(* IEC 61131-3 sources: Universal/UNIVERSAL/Interfaces/UNIVERSAL/Device1/Terminal1 (part 2) *)

FUNCTION Upgrade_1_ENTER
	// Upgrade.En_Read:= TRUE;
    Upgrade.Check_Upgrade:= TRUE;
END_FUNCTION

FUNCTION Upgrade_1_PRG
    IF (Upgrade.En_FirmWare) THEN
        Upgrade.En_Upgrade:= TRUE;
        GotoMask(Upgrade_Progress);
    ELSE
        Upgrade_1_ENTER();
    END_IF;
END_FUNCTION

(*				BEGIN IMPORT CODE				*)

FUNCTION NetMap_ENTER

    CurSlave:=      CurPosition;
    CurSlaveShow:=  TRUE;   // сообщаем стратегии что сейчас будем показывать текущего ведомого

	GotoMaskID(32); //SlaveState

END_FUNCTION

FUNCTION SlaveState_ESC
    CurSlaveShow:=  FALSE;// сообщаем стратегии что прекращаем показывать текущего ведомого
    IF (GetAlarmsCount() > 0) THEN
        SetLedStatus(12,1);// возвращаем управление колокольчиком основной программе
    ELSE
        SetLedStatus(12,0);
    END_IF;
    GotoMask(NetMap);
END_FUNCTION

FUNCTION Incr_REAL_x1000
    __TMP_REAL := __TMP_REAL + TO_REAL(__SYSVA_KEY_COUNTER)*1000.0;
    CheckLimitsDecr();
END_FUNCTION

FUNCTION Decr_REAL_x1000
    __TMP_REAL := __TMP_REAL - TO_REAL(__SYSVA_KEY_COUNTER)*1000.0;
    CheckLimitsDecr();
END_FUNCTION

(*				END IMPORT CODE					*)

FUNCTION DeviceRole_Class_PRG
    IF (StatePRG = STATE_PRG_READY) THEN
        StoreMask();
        StatePRG:= STATE_PRG_ON;
        NextCycleAction:= 2;
    ELSIF (StatePRG = STATE_PRG_ON) THEN
        Compare();
        IF (temp_Role <> Role) THEN
            IF (temp_Role = 0)OR(Role_Master) THEN
                (*Reboot_Reason:= 3;// изменение роли устройства
                StoreMask();
                GotoMask(NeedReboot);*)
                ShowPopUpQuestion(4); // изменение роли устройства
            ELSE
                Role:=      temp_Role;
                StoreMask();
                StatePRG:= STATE_PRG_READY;
                NextCycleAction:=   1;
            END_IF;
        ELSE
            StoreMask();
            StatePRG:= STATE_PRG_READY;
            NextCycleAction:=   1;
        END_IF;
    END_IF;
END_FUNCTION

FUNCTION DeviceRole_Class_ENTER
    IF (StatePRG <> STATE_PRG_READY) THEN
	    Compare();
        IF (temp_Role <> Role) THEN
            IF (temp_Role = 0)OR(Role_Master) THEN
                ShowPopUpQuestion(4);// изменение роли устройства
            ELSE
                Role:=  temp_Role;
            END_IF;
        END_IF;
    END_IF;
END_FUNCTION

FUNCTION HeatType_ENTER
	Compare ();
    IF (temp_HeatType <> HeatType) THEN
        IF (temp_HeatType = 1) OR (HeatType = 1)  THEN
            ShowPopUpQuestion(3);// изменение типа нагрева
        ELSE
            HeatType:= temp_HeatType;
        END_IF;
    END_IF;
END_FUNCTION

// Тест. Управление частотником
FUNCTION Main_Testing_ESC
    IF (EnPwdChgM) THEN
	    En_Testing:= TRUE;
        GotoLoop(TESTING);
        StatePRG:= STATE_PRG_READY;
    END_IF;
END_FUNCTION

FUNCTION Testing_ESC
    En_Testing:= FALSE;
	GotoMain();
    StatePRG:= STATE_PRG_OFF;
END_FUNCTION

// ModBus
FUNCTION Show_ports
    IF (Temp_MB_port = 0) THEN
        En_MB_Ethernet:= FALSE;
        En_MB_BMS_Card:= FALSE;
        En_MB_BMS2:= FALSE;
        En_MB_BMS:= FALSE;
    ELSIF (Temp_MB_port = 1) THEN
        En_MB_Ethernet:= TRUE;
        En_MB_BMS_Card:= FALSE;
        En_MB_BMS2:= FALSE;
        En_MB_BMS:= FALSE;
    ELSIF (Temp_MB_port = 2) THEN
        En_MB_Ethernet:= FALSE;
        En_MB_BMS_Card:= TRUE;
        En_MB_BMS2:= FALSE;
        En_MB_BMS:= TRUE;
        Temp_MB_Baudrate:= BMS_Card.Baudrate;
        Temp_MB_StopBits:= BMS_Card.StopBits;
        Temp_MB_Parity:= BMS_Card.Parity;
    ELSIF (Temp_MB_port = 3) THEN
        En_MB_Ethernet:= FALSE;
        En_MB_BMS_Card:= FALSE;
        En_MB_BMS2:= TRUE;
        En_MB_BMS:= TRUE;
        Temp_MB_Baudrate:= BMS2.Baudrate;
        Temp_MB_StopBits:= BMS2.StopBits;
        Temp_MB_Parity:= BMS2.Parity;
    END_IF;
END_FUNCTION

FUNCTION Port_Sel_ENTER
    IF (Temp_MB_port <> TO_USINT(__TMP_BYTE)) THEN
        Compare();
	    Show_ports();
    ELSE
        GotoNextField();
    END_IF;
END_FUNCTION

FUNCTION MB_Settings_1_PRG
    IF (StatePRG = STATE_PRG_READY) THEN
        StoreMask();
        StatePRG:= STATE_PRG_ON;
        NextCycleAction:=   1;
    ELSIF (StatePRG = STATE_PRG_ON) THEN
        Compare();
        IF (Temp_MB_port <> MB_port)
            OR (Temp_MB_Address <> MB_Address)
            OR ((Temp_MB_port = 2)AND (Temp_MB_Baudrate <> BMS_Card.Baudrate))
            OR ((Temp_MB_port = 2)AND (Temp_MB_StopBits <> BMS_Card.StopBits))
            OR ((Temp_MB_port = 2)AND (Temp_MB_Parity <> BMS_Card.Parity))
            OR ((Temp_MB_port = 3)AND (Temp_MB_Baudrate <> BMS2.Baudrate))
            OR ((Temp_MB_port = 3)AND (Temp_MB_StopBits <> BMS2.StopBits))
            OR ((Temp_MB_port = 3)AND (Temp_MB_Parity <> BMS2.Parity))
            THEN
            (*Reboot_Reason:= 4;// изменение настроек ModBus
            StoreMask();
            GotoMask(NeedReboot);*)
            ShowPopUpQuestion(5);// изменение настроек ModBus
        ELSE
            Show_ports();
            StatePRG:= STATE_PRG_READY;
            NextCycleAction:=   1;
        END_IF;
    END_IF;
END_FUNCTION

FUNCTION MB_Settings_1_ESC
    IF (StatePRG = STATE_PRG_READY) THEN
        GlobalEsc();
    ELSIF (StatePRG = STATE_PRG_ON) THEN
        Compare();
        IF (Temp_MB_port <> MB_port)
            OR (Temp_MB_Address <> MB_Address)
            OR ((Temp_MB_port = 2)AND (Temp_MB_Baudrate <> BMS_Card.Baudrate))
            OR ((Temp_MB_port = 2)AND (Temp_MB_StopBits <> BMS_Card.StopBits))
            OR ((Temp_MB_port = 2)AND (Temp_MB_Parity <> BMS_Card.Parity))
            OR ((Temp_MB_port = 3)AND (Temp_MB_Baudrate <> BMS2.Baudrate))
            OR ((Temp_MB_port = 3)AND (Temp_MB_StopBits <> BMS2.StopBits))
            OR ((Temp_MB_port = 3)AND (Temp_MB_Parity <> BMS2.Parity))
            THEN
            (*Reboot_Reason:= 4;// изменение настроек ModBus
            StoreMask();
            GotoMask(NeedReboot);*)
            ShowPopUpQuestion(5);// изменение настроек ModBus
        ELSE
            GlobalEsc();
        END_IF;
    END_IF;
END_FUNCTION

FUNCTION Mul_DWORD_x2
    __TMP_DWORD := __TMP_DWORD * 2;
    CheckLimitsIncr();
END_FUNCTION

FUNCTION Div_DWORD_x2
    __TMP_DWORD := __TMP_DWORD / 2;
    CheckLimitsDecr();
END_FUNCTION
FUNCTION Upgrade_OS_ESC
	Upgrade.REQ_OS_upgrade:= FALSE;
    GotoLoop(UPGRADE);
END_FUNCTION

FUNCTION Upgrade_OS_PRG
	Upgrade.ANSW_OS_upgrade:= TRUE;
    GotoMask(Upgrade_Progress);
END_FUNCTION

FUNCTION PRG_button_goto10
	 IF (StatePRG = STATE_PRG_READY) THEN
        StoreMask();
        StatePRG:= STATE_PRG_ON;
        NextCycleAction:=   2;
    ELSIF (StatePRG = STATE_PRG_ON) THEN
        Compare();
        StatePRG:= STATE_PRG_READY;
        NextCycleAction:=   1;
    END_IF;
END_FUNCTION

// Переход на следующую маску в режиме программирования
FUNCTION DOWN_ENTER_Move
    IF (StatePRG = STATE_PRG_ON) THEN
        GotoNextMask();
        checkZeroColumn:= TRUE;
    END_IF;
END_FUNCTION

// Переход на предыдущую маску в режиме программирования
FUNCTION UP_ENTER_Move
    IF (StatePRG = STATE_PRG_ON) THEN
        GotoPreviousMask();
        checkZeroColumn:= TRUE;
    END_IF;
END_FUNCTION

FUNCTION Decrement // уменьшение байтовой переменной с индикацией стрелки
    Decrement_BYTE();
    downArrow:= TRUE;
END_FUNCTION

FUNCTION Increment  // увеличение байтовой переменной с индикацией стрелки
    Increment_BYTE();
    upArrow:=   TRUE;
END_FUNCTION

FUNCTION BoolDown   // уменьшение булевой переменной с индикацией стрелки
	BoolSwap();
    downArrow:= TRUE;
END_FUNCTION

FUNCTION BoolUp     // увеличение булевой переменной с индикацией стрелки
	BoolSwap();
    upArrow:=   TRUE;
END_FUNCTION

//FUNCTION FConfigSetBool  // принятие булевой переменной с индикацией выбора
    //MakeChoice:=        TRUE;
    //NextCycleAction:=   3;
//END_FUNCTION
//
//FUNCTION FConfigSetByte  // принятие байтовой переменной с индикацией выбора
    //Compare();
    //MakeChoice:=        TRUE;
    //NextCycleAction:=   3;
//END_FUNCTION
//
//FUNCTION FConfigSetPriority  // принятие  переменной ModeSEQ c переходом к петле CONFIRM_CONFIG
    //Compare();
    //NextCycleAction:=   6;
//END_FUNCTION
//
//
//FUNCTION FConfig_LastMask    // принятие последней в петле байтовой переменной с индикацией выбора
	//Compare();
    //MakeChoice:=        TRUE;
    //IF (IsPOOL) THEN
        //NextCycleAction:=   6;
    //ELSE
        //NextCycleAction:=   5;
    //END_IF;
//END_FUNCTION
//
//FUNCTION FConfig_ESC  // запрос на возврат к началу первой конфигурации
    //IF (CompletePreConfig) THEN
        //ShowPopUpQuestion(12);  // Выйти из мастера конфигураций
    //ELSE
        //StatePRG:= STATE_PRG_ALWAYS_ON;
        //MakeChoice:=    FALSE;
        //ShowPopUpQuestion(7);   // Вернуться к началу конфигурации?
    //END_IF;
//END_FUNCTION

FUNCTION SWAP_Sp100
    BoolSwap();
    IF (wCoil_Mode_A_B)AND(Par_Sp100) THEN
        ShowPopUpMessage(12, SHORT_POPUP_TIME);
        //Par_Sp100:=   FALSE;
    END_IF;
END_FUNCTION

FUNCTION SWAP_Tp10 // Проверка при переключении параметра Tp10 в меню
    BoolSwap();
    IF NOT(SNSR_Thru.Use)OR(SNSR_Thru.Error <> 10) THEN
		IF NOT(Par_Tp10)THEN
            ShowPopUpMessage(11, SHORT_POPUP_TIME);
            Par_Tp10:=   TRUE;
        END_IF;
    END_IF;
END_FUNCTION

FUNCTION ManualManager // Вход и выход из ручного режима
    VAR_INPUT
        in : BOOL;
    END_VAR

    IF (in)AND NOT(ManualManage)THEN
        ManualManage:=  TRUE;
        ShowPopUpMessage(15, SHORT_POPUP_TIME); //  Ручной режим включен
    ELSIF NOT(in)AND (ManualManage)THEN
        ManualManage:=  FALSE;
        CurRow:= 0;
        ShowPopUpMessage(16, SHORT_POPUP_TIME); // Ручной режим выключен
    END_IF;

END_FUNCTION

FUNCTION Param_UP   // Переход вверх

    IF (StatePRG = STATE_PRG_READY) THEN
        IF (CurRow > 1) THEN
            CurRow:= CurRow - 1;
        ELSE

            //MaskMng.shift_position:= -(TO_DINT(__SYSVA_KEY_COUNTER)/20) - 1;
            Position:= Position - TO_DINT(__SYSVA_KEY_COUNTER)/20 - 1;

            //IF (Position + MaskMng.shift_position < 1) THEN
                //__SYSVA_KEY_COUNTER:= 0;
                //CurRow:= num_Rows;
                //Beep();
            //END_IF;
            IF (Position < 1) THEN
                __SYSVA_KEY_COUNTER:= 0;
                Position:= cnt_Items - num_Rows + 1;
                CurRow:= num_Rows;
                //Beep();
            END_IF;
        END_IF;
        CurList_Position:= Position + CurRow - 1;
        Display.Hint:= Display.Descr[CurRow];
        update_ParamMenu_List:=      TRUE;
    ELSIF (StatePRG = STATE_PRG_ON) THEN

        CASE (Display.value_Storage[CurRow_modePRG]) OF
            0: // BOOL
                IF (Display.value_BOOL[CurRow_modePRG] = 2) THEN
                    Display.value_BOOL[CurRow_modePRG]:= 1;
                END_IF;
            1: // UINT
                Display.value_INT[CurRow_modePRG]:=  Display.value_INT[CurRow_modePRG] + TO_INT(__SYSVA_KEY_COUNTER);
            2: // REAL
                Display.value_REAL[CurRow_modePRG]:=  Display.value_REAL[CurRow_modePRG] + TO_REAL(__SYSVA_KEY_COUNTER)/10.0;
        END_CASE;
        CheckValueBorders ();
    END_IF;
    NextCycleAction:= 12; //Обновление подсказки и позиции
END_FUNCTION

FUNCTION Param_DOWN   // Переход вверх

    IF (StatePRG = STATE_PRG_READY) THEN
        IF (CurRow < num_Rows) THEN
            CurRow:= CurRow + 1;
        ELSE
            Position:= Position + TO_DINT(__SYSVA_KEY_COUNTER)/20 + 1;

            IF (Position > cnt_Items - num_Rows + 1) THEN
                __SYSVA_KEY_COUNTER:= 0;
                Position:= 1;
                CurRow:= 1;
                //Beep();
            END_IF;
           //MaskMng.shift_position:= TO_DINT(__SYSVA_KEY_COUNTER)/20 + 1;
            //
            //IF (Position + MaskMng.shift_position > cnt_Items - num_Rows + 1) THEN
                //__SYSVA_KEY_COUNTER:= 0;
                //CurRow:= 1;
                //Beep();
            //END_IF;
        END_IF;
        CurList_Position:= Position + CurRow - 1;
        Display.Hint:= Display.Descr[CurRow];
        update_ParamMenu_List:=      TRUE;
    ELSIF (StatePRG = STATE_PRG_ON) THEN

        CASE (Display.value_Storage[CurRow_modePRG]) OF
            0: // BOOL
                IF (Display.value_BOOL[CurRow_modePRG] = 1) THEN
                    Display.value_BOOL[CurRow_modePRG]:= 2;
                END_IF;
            1: // UINT
                Display.value_INT[CurRow_modePRG]:=  Display.value_INT[CurRow_modePRG] - TO_INT(__SYSVA_KEY_COUNTER);
            2: // REAL
                Display.value_REAL[CurRow_modePRG]:=  Display.value_REAL[CurRow_modePRG] - TO_REAL(__SYSVA_KEY_COUNTER)/10.0;
        END_CASE;
        CheckValueBorders ();
    END_IF;
    NextCycleAction:= 12; //Обновление подсказки и позиции
END_FUNCTION

FUNCTION Param_ENTER   // Подтверждение
    IF (StatePRG = STATE_PRG_ON) THEN

        Write_Parameter();

        IF (CurRow_modePRG < num_Rows) THEN
            CurRow_modePRG:= CurRow_modePRG + 1;
        ELSE
            Position:= Position + TO_DINT(__SYSVA_KEY_COUNTER)/20 + 1;

            IF (Position > cnt_Items - num_Rows + 1) THEN
                __SYSVA_KEY_COUNTER:= 0;
                Position:= 1;
                CurRow_modePRG:= 1;
                //Beep();
            END_IF;
        END_IF;
        //getParamMenu:=      TRUE;
        CurList_Position:= Position + CurRow_modePRG - 1;
        Display.Hint:= Display.Descr[CurRow_modePRG];
        update_ParamMenu_List:=      TRUE;
    END_IF;

    NextCycleAction:= 12; //Обновление подсказки и позиции
END_FUNCTION

FUNCTION Write_Parameter // Запись параметра

    CheckValueBorders ();
    CASE (Display.value_Storage[CurRow_modePRG]) OF
        0: // BOOL
            IF (Display.value_BOOL[CurRow_modePRG] = 1) THEN ;
                param.BOOL[Display.value_Address[CurRow_modePRG]]:= TRUE;
            ELSIF (Display.value_BOOL[CurRow_modePRG] = 2) THEN ;
                param.BOOL[Display.value_Address[CurRow_modePRG]]:= FALSE;
            END_IF;
        1: // INT
            IF (param.INT[Display.value_Address[CurRow_modePRG]] <>
                Display.value_INT[CurRow_modePRG])
            THEN
                //MaskMng.param_ChangeNotify:= Display.Descr[CurRow_modePRG];
                param.INT[Display.value_Address[CurRow_modePRG]]:= Display.value_INT[CurRow_modePRG];
            END_IF;
        2: // REAL
            IF (param.REAL[Display.value_Address[CurRow_modePRG]] <>
                Display.value_REAL[CurRow_modePRG])
            THEN
                //MaskMng.param_ChangeNotify:= Display.Descr[CurRow_modePRG];
                param.REAL[Display.value_Address[CurRow_modePRG]]:= Display.value_REAL[CurRow_modePRG];
            END_IF;
    END_CASE;

    MaskMng.param_ChangeNotify:= TO_USINT(Display.Descr[CurRow_modePRG]);
END_FUNCTION

FUNCTION Param_ESC   // Переход вверх

    IF (StatePRG = STATE_PRG_READY) THEN
        //cnt_Items:=  0;
        Position:=      1;
        autoHideArrowsOff:=     FALSE;
        GlobalEsc();
    ELSIF (StatePRG = STATE_PRG_ON) THEN
        StatePRG:=  STATE_PRG_READY;
        CurRow:= CurRow_modePRG;
        CurRow_modePRG:=    0;
        //getParamMenu:=      TRUE;
        update_ParamMenu_List:= TRUE;
    END_IF;

END_FUNCTION

FUNCTION CheckValueBorders   // Проверка границ значений

    CASE (Display.value_Storage[CurRow_modePRG]) OF
            0: // BOOL
               ;
            1: // UINT
                IF (Display.value_INT[CurRow_modePRG] < Display.value_MinINT[CurRow_modePRG]) THEN
                    Display.value_INT[CurRow_modePRG]:= Display.value_MaxINT[CurRow_modePRG];
                    Beep();
                ELSIF (Display.value_INT[CurRow_modePRG] > Display.value_MaxINT[CurRow_modePRG]) THEN
                    Display.value_INT[CurRow_modePRG]:= Display.value_MinINT[CurRow_modePRG];
                    Beep();
                END_IF;
            2: // REAL
                IF (Display.value_REAL[CurRow_modePRG] < Display.value_MinREAL[CurRow_modePRG]) THEN
                    Display.value_REAL[CurRow_modePRG]:= Display.value_MaxREAL[CurRow_modePRG];
                    Beep();
                ELSIF (Display.value_REAL[CurRow_modePRG] > Display.value_MaxREAL[CurRow_modePRG]) THEN
                    Display.value_REAL[CurRow_modePRG]:= Display.value_MinREAL[CurRow_modePRG];
                    Beep();
                END_IF;
        END_CASE;
END_FUNCTION

FUNCTION UpdateCurPos
// Отображение расширенного описания текущей позиции
    IF (ModePRG) THEN
        Display.Hint:= Display.Descr[CurRow_modePRG];
        CurList_Position:= Position + CurRow_modePRG - 1;
    ELSE
        Display.Hint:= Display.Descr[CurRow];
        CurList_Position:= Position + CurRow - 1;
    END_IF;
END_FUNCTION

FUNCTION CheckListBorders   // Проверка границ списка
    //VAR
        //lastPixelPosition : USINT; // позиция последнего пикселя
    //END_VAR;
//
    //IF (Position <= 1) THEN
        //upArrow:= FALSE;
    //ELSE
        //upArrow:= TRUE;
    //END_IF;
//
    //IF (Position >= cnt_Items - num_Rows + 1) OR
       //(cnt_Items < num_Rows)
    //THEN
        //downArrow:= FALSE;
    //ELSE
        //downArrow:= TRUE;
    //END_IF;

(*
    IF (Slider_Height = 0) THEN
        Slider_Height:= TO_USINT(48 / cnt_Items);
    END_IF;

    lastPixelPosition:= Slider_Height * TO_USINT(Position);

    IF (lastPixelPosition <= 8) THEN
        Slider_1:= lastPixelPosition;
    ELSIF (lastPixelPosition <= 16) THEN
        Slider_2:= lastPixelPosition - 8;
        IF (Slider_Height > 8) THEN
             Slider_1:= 16 - (Slider_Height - (16 - lastPixelPosition)) ;
        END_IF;
    END_IF;
*)
END_FUNCTION

FUNCTION Param_PRG   //

    //StoreMask();

    IF (StatePRG = STATE_PRG_READY) THEN        // вход в режим редактирования
            //150121 2.7.6.0 Запрет для пользователя упразднен, т.к. скрываются все ненужные пункты меню.
            //IF (UnitOn)AND(PwdTyp < 2) THEN         //  Для пользователя изменения во время работы запрещены
            //    ShowPopUpMessage(1, POPUP_TIME);    //  Выключите установку для изменения настроек!
            //ELSE
                StatePRG:=  STATE_PRG_ON;
                CurRow_modePRG:= CurRow;
                CurRow:=    0;
                // getParamMenu:=      TRUE;
                update_ParamMenu_List:= TRUE;
                NextCycleAction:= 12; //Обновление подсказки и позиции
            //END_IF;

    ELSIF (StatePRG = STATE_PRG_ON) THEN        // выход из режима редактирования

        Write_Parameter();

        StatePRG:=  STATE_PRG_READY;
        CurRow:= CurRow_modePRG;
        CurRow_modePRG:=    0;
        //getParamMenu:=      TRUE;
        update_ParamMenu_List:= TRUE;
        NextCycleAction:= 12; //Обновление подсказки и позиции
    END_IF;
END_FUNCTION

//FUNCTION GoToConfiguration
	////load_Config:= TRUE;
    ////isConfigMenu:= TRUE;
    ////getConfigMenu:= TRUE;
    ////CurRow:=            1;
    ////CurRow_modePRG:=    0;
    ////cnt_Items:= 0;
    ////GotoMask(LoadConfig_Mask);
    //ConfigMng.checkConfigFile:= TRUE;
//END_FUNCTION

FUNCTION ConfigMenu_UP   // Переход вверх
    IF (CurRow > 1) THEN
        CurRow:= CurRow - 1;
    ELSE
        Position:= Position - TO_DINT(__SYSVA_KEY_COUNTER)/20 - 1;

        IF (Position < 1) THEN
            __SYSVA_KEY_COUNTER:= 0;
            Position:= cnt_Items - num_Rows + 1;
            CurRow:= num_Rows;
            //Beep();
        END_IF;

        IF (isConfigMenu) THEN
            getConfigMenu:= TRUE;
        ELSE
            getParamMenu:= TRUE;
        END_IF;
    END_IF;

    CurList_Position:= Position + CurRow - 1;
    Display.Hint:= Display.Descr[CurRow];
END_FUNCTION

FUNCTION ConfigMenu_DOWN   // Переход вниз
    IF (CurRow < num_Rows) THEN
        CurRow:= CurRow + 1;
    ELSE
        Position:= Position + TO_DINT(__SYSVA_KEY_COUNTER)/20 + 1;

        IF (Position > cnt_Items - num_Rows + 1) THEN
            __SYSVA_KEY_COUNTER:= 0;
            Position:= 1;
            CurRow:= 1;
            //Beep();
        END_IF;

        IF (isConfigMenu) THEN
            getConfigMenu:= TRUE;
        ELSE
            getParamMenu:= TRUE;
        END_IF;
    END_IF;

    CurList_Position:= Position + CurRow - 1;
    Display.Hint:= Display.Descr[CurRow];
END_FUNCTION

FUNCTION ConfigMenu_ENTER   //
    IF (Display.value_BOOL[CurRow] = 4) // каталог
    THEN
        //IF (CurLevel < 10) THEN
            //Display.Path.MenuPoint[CurLevel]:= CurMenuPoint;
            //Display.Path.Position[CurLevel]:= Position;
            //Display.Path.Row[CurLevel]:= CurRow;
            //CurLevel:= CurLevel + 1;
            SaveMenuPos();
            CurMenuPoint:= TO_DINT(Display.Descr[CurRow]);
            getConfigMenu:= TRUE;
        //END_IF;
        IF (CurLevel < 10) THEN
            CurRow:=            1;
            Position:=          1;
            CurList_Position:=  1;
        END_IF;
    ELSIF (Display.value_BOOL[CurRow] = 7) // действие?
    THEN
        //Display.Path.MenuPoint[CurLevel]:= CurMenuPoint;
        //Display.Path.Position[CurLevel]:= Position;
        //Display.Path.Row[CurLevel]:= CurRow;
        SaveMenuPos();
        CurMenuPoint:= TO_DINT(Display.Descr[CurRow]);
        getConfigMenu:= TRUE;
    ELSE
        Display.Path.MenuPoint[CurLevel]:= CurMenuPoint;
        Display.Path.Position[CurLevel]:= Position;
        Display.Path.Row[CurLevel]:= CurRow;
        CurMenuPoint:= TO_DINT(Display.Descr[CurRow]);
        setConfigItem:= TRUE;
    END_IF;
    //NextCycleAction:= 12;
    Display.Hint:= Display.Descr[CurRow];
END_FUNCTION

FUNCTION ConfigMenu_ESC   //
    IF (CurLevel > ConfigStartLevel) THEN
        LoadMenuPos();
    ELSE
        //Перебрасываем в начало конфигуратора
        Position:=          1;
        CurMenuPoint:=      0;
        CurList_Position:=  1;
        CurRow:=            1;

        //IF (CurMenuPoint <> 0) THEN
            //Position:= 1;
            //CurMenuPoint:= 0;
            //CurList_Position:= 1;
            //CurRow:= 1;
        //ELSE
            //IF (ConfigStartLevel <> 0) THEN
                //IF (IsConfigChanged) THEN
                    ////Сохранить конфигурацию?
                    //ShowPopUpQuestion(21); //InstantAction:=  255; //DF_CFG_END
                //ELSE
                    //GlobalEsc();
                //END_IF;
            //END_IF;
        //END_IF;
    END_IF;

    getConfigMenu:= TRUE;
    //cnt_Items:=  0;

    //NextCycleAction:= 12;
END_FUNCTION

FUNCTION Signal_DOWN

    CASE CurRow OF
        1:
            mask_List_pos:=  mask_List_pos + TO_DINT(__SYSVA_KEY_COUNTER)/20 + 1;

            IF (mask_List_pos > cnt_Items) THEN
                __SYSVA_KEY_COUNTER:= 0;
                mask_List_pos:= 1;
                Beep();
            END_IF;

            Display.Descr[1]:= mask_List[mask_List_pos];
            Display.Hint:= mask_List_Sec[mask_List_pos];
            //Display.Hint:= Display.Descr[1];
            ConfigMng.recount_Types:= TRUE;
            recount_IO:= TRUE;
            getMinMax:= TRUE;

        2:
           (*Сдвиг окна позиции*)
			ConfigMng.mask_IO_List_pos:= ConfigMng.mask_IO_List_pos + TO_DINT(__SYSVA_KEY_COUNTER)/20 + 1;
			(*Проверка выхода за границы*)
			IF (ConfigMng.mask_IO_List_pos > ConfigMng.cnt_IO_Items) THEN
                __SYSVA_KEY_COUNTER:= 0;
                ConfigMng.mask_IO_List_pos:= 0;
                Beep();
            END_IF;

			Display.Descr[2]:= TO_UINT(ConfigMng.mask_IO_List[ConfigMng.mask_IO_List_pos]);
            //Display.Descr[3]:= TO_USINT(ConfigMng.mask_IO_List_pos);
            //IF (ConfigMng.mask_IO_List_pos = 0) THEN
                //Display.Hint:= 0;
            //ELSE
                //Display.Hint:= ConfigMng.mask_IO_List[0] + 1;
            //END_IF;

        3:
            (*Сдвиг окна позиции*)
			ConfigMng.mask_TypeList_pos:= ConfigMng.mask_TypeList_pos - TO_DINT(__SYSVA_KEY_COUNTER)/20 - 1;
			(*Проверка выхода за границы*)
			IF (ConfigMng.mask_TypeList_pos < 0) THEN
                __SYSVA_KEY_COUNTER:= 0;
                ConfigMng.mask_TypeList_pos:= ConfigMng.cnt_TypeItems - 1;
                Beep();
            END_IF;

			Display.Descr[3]:= TO_UINT(ConfigMng.mask_TypeList[ConfigMng.mask_TypeList_pos]);

        4:
            Display.value_REAL[4]:= Display.value_REAL[4] - TO_REAL(__SYSVA_KEY_COUNTER/20) - 1.0;
            IF (Display.value_REAL[4] < Display.value_MinREAL[4]) THEN
                Display.value_REAL[4]:= Display.value_MaxREAL[4];
                Beep();
            END_IF;

        5:
            Display.value_REAL[5]:= Display.value_REAL[5] - TO_REAL(__SYSVA_KEY_COUNTER/20) - 1.0;
            IF (Display.value_REAL[5] < Display.value_MinREAL[5]) THEN
                Display.value_REAL[5]:= Display.value_MaxREAL[5];
                Beep();
            END_IF;
    END_CASE;
END_FUNCTION

FUNCTION Signal_UP

    CASE CurRow OF
        1:
            mask_List_pos:=  mask_List_pos - TO_DINT(__SYSVA_KEY_COUNTER)/20 - 1;

            IF (mask_List_pos < 1) THEN
                __SYSVA_KEY_COUNTER:= 0;
                mask_List_pos:= cnt_Items;
                Beep();
            END_IF;
            //getIOConfig:= TRUE;

            Display.Descr[1]:= mask_List[mask_List_pos];
            Display.Hint:= mask_List_Sec[mask_List_pos];
            //Display.Descr[2]:= ConfigMng.mask_IO_List[0];
            //Display.Hint:= Display.Descr[1];
            ConfigMng.recount_Types:= TRUE;
            recount_IO:= TRUE;
            getMinMax:= TRUE;

        2:
           (*Сдвиг окна позиции*)
			ConfigMng.mask_IO_List_pos:= ConfigMng.mask_IO_List_pos - TO_DINT(__SYSVA_KEY_COUNTER)/20 - 1;
			(*Проверка выхода за границы*)
			IF (ConfigMng.mask_IO_List_pos < 0) THEN
                __SYSVA_KEY_COUNTER:= 0;
                ConfigMng.mask_IO_List_pos:= ConfigMng.cnt_IO_Items;
                Beep();
            END_IF;

			Display.Descr[2]:= TO_UINT(ConfigMng.mask_IO_List[ConfigMng.mask_IO_List_pos]);
            //Display.Descr[3]:= TO_USINT(ConfigMng.mask_IO_List_pos);
            //IF (ConfigMng.mask_IO_List_pos = 0) THEN
                //Display.Hint:= 0;
            //ELSE
                //Display.Hint:= ConfigMng.mask_IO_List[0] + 1;
            //END_IF;

        3:
            (*Сдвиг окна позиции*)
			ConfigMng.mask_TypeList_pos:= ConfigMng.mask_TypeList_pos + TO_DINT(__SYSVA_KEY_COUNTER)/20 + 1;
			(*Проверка выхода за границы*)
			IF (ConfigMng.mask_TypeList_pos > ConfigMng.cnt_TypeItems - 1) THEN
                __SYSVA_KEY_COUNTER:= 0;
                ConfigMng.mask_TypeList_pos:= 0;
                Beep();
            END_IF;

			Display.Descr[3]:= TO_UINT(ConfigMng.mask_TypeList[ConfigMng.mask_TypeList_pos]);

        4:
            Display.value_REAL[4]:= Display.value_REAL[4] + TO_REAL(__SYSVA_KEY_COUNTER/20) + 1.0;
            IF (Display.value_REAL[4] > Display.value_MaxREAL[4]) THEN
                Display.value_REAL[4]:= Display.value_MinREAL[4];
                Beep();
            END_IF;

        5:
            Display.value_REAL[5]:= Display.value_REAL[5] + TO_REAL(__SYSVA_KEY_COUNTER/20) + 1.0;
            IF (Display.value_REAL[5] > Display.value_MaxREAL[5]) THEN
                Display.value_REAL[5]:= Display.value_MinREAL[5];
                Beep();
            END_IF;

    END_CASE;
END_FUNCTION

FUNCTION Signal_ESC

    //RestoreMask();
    GlobalEsc();

    //CurLevel:= CurLevel - 1;
    //CurMenuPoint:=  Display.Path.MenuPoint[CurLevel];
    //Position:= Display.Path.Position[CurLevel];
    //CurRow:= Display.Path.Row[CurLevel];
    //Display.Path.MenuPoint[CurLevel]:= 0;
    //CurList_Position:= Position + CurRow - 1;

    //getConfigMenu:= TRUE;

END_FUNCTION

FUNCTION Signal_ENTER

    CASE CurRow OF
        1:
            recount_IO:= TRUE;
            //IF (ConfigMng.mask_IO_List_pos = 0) THEN
                //Display.Hint:= 0;
            //ELSE
                //Display.Hint:= ConfigMng.mask_IO_List[0] + 1;
            //END_IF;

            IF (num_Rows = 2) THEN
                CurRow:= 2;
            ELSE
                CurRow:= 3;
                Display.Descr[3]:= TO_UINT(ConfigMng.mask_TypeList[ConfigMng.mask_TypeList_pos]);
            END_IF;
        2:
            ConfigMng.setIoItem:= TRUE;
            //Display.Hint:= 0;
            CurRow:= 1;
        3:
            recount_IO:= TRUE;
            CASE Display.Descr[3] OF
                5,6,7,8,9: //AI с min/max
                    CurRow:= 4;
            ELSE
                CurRow:= 2;
            END_CASE;
            getMinMax:= TRUE;
        4:
            //сделать запись в переменную Min для сигнала
            ConfigMng.setMinMax:= TRUE;
            CurRow:= 5;
        5:
            //сделать запись в переменную Max для сигнала
            ConfigMng.setMinMax:= TRUE;
            CurRow:= 2;
    END_CASE;

END_FUNCTION

// Управление маской Control_Mode------------
FUNCTION Control_Mode_UP
	upArrow:= TRUE;
    IF (temp_Mode_Control > 1) THEN
        temp_Mode_Control:= temp_Mode_Control - 1;
    ELSE
        temp_Mode_Control:= 10;
    END_IF;

    IF (IsPOOL)(*OR(IsICE)*) THEN
        IF (temp_Mode_Control = 10) THEN
            temp_Mode_Control:= 8;
        ELSIF (temp_Mode_Control = 6) OR (temp_Mode_Control = 5) THEN
            temp_Mode_Control:= 4;
        ELSIF (temp_Mode_Control = 3) THEN
            temp_Mode_Control:= 2;
        END_IF;
    END_IF;
END_FUNCTION

FUNCTION Control_Mode_DOWN
	downArrow:= TRUE;
    IF (temp_Mode_Control < 10) THEN
        temp_Mode_Control:= temp_Mode_Control + 1;
    ELSE
        temp_Mode_Control:= 1;
    END_IF;

    IF (IsPOOL)(*OR(IsICE)*) THEN
        IF (temp_Mode_Control = 3) THEN
            temp_Mode_Control:= 4;
        ELSIF (temp_Mode_Control = 5) OR (temp_Mode_Control = 6) THEN
            temp_Mode_Control:= 7;
        ELSIF (temp_Mode_Control = 9) OR (temp_Mode_Control = 10) THEN
            temp_Mode_Control:= 1;
        END_IF;
    END_IF;
END_FUNCTION

FUNCTION Control_Mode_ENTER
	Mode_Control:= temp_Mode_Control;
END_FUNCTION
//-------------------------------------------

// Управление маской Schedule_Manage------------
FUNCTION Schedule_Manage_UP
	upArrow:= TRUE;
    temp_En_Schedule:= NOT(temp_En_Schedule);
END_FUNCTION

FUNCTION Schedule_Manage_DOWN
	downArrow:= TRUE;
    temp_En_Schedule:= NOT(temp_En_Schedule);
END_FUNCTION

FUNCTION Schedule_Manage_ENTER
	En_Schedule:= temp_En_Schedule;
END_FUNCTION

//-------------------------------------------

//FUNCTION Load_Config
    //load_Config:= TRUE;
    //GotoMask(LoadConfig_Mask);
//END_FUNCTION

// Управление масками вх/вых -------------------------------------
FUNCTION IO_DOWN
    IF (StatePRG = STATE_PRG_ON) THEN
        IF (CurRow = 3) THEN // Надпись Режим
            IF (Display.value_BOOL[1] = 1) THEN //руч.
                CurRow:= 4;
            ELSE
                IF  (Display.MaskID = 11) OR // Дискретные входы
                    (Display.MaskID = 14)    // Аналоговые выходы
                THEN
                    CurRow:= 5;
                ELSE
                    Beep();
                END_IF;
            END_IF;
        ELSIF (CurRow = 4) THEN // Надпись Статус
            CurRow:= 3;
        ELSIF (CurRow = 5) THEN // Надпись инверсия
            CurRow:= 3;
        ELSIF (CurRow_modePRG = 3) THEN // Изменение режима
            IF (Display.value_BOOL[1] = 0) THEN
                 Display.value_BOOL[1]:= 1;
            ELSIF( Display.value_BOOL[1] = 1) THEN
                Display.value_BOOL[1]:= 0;
            END_IF;
            //MaskMng.ValueWasChanged:= TRUE;
        ELSIF (CurRow_modePRG = 4) THEN // Изменение значения
            CASE Display.MaskID OF
                11, 13:(*Digital*)
                    Display.value_BOOL[2]:= 2; //OFF
                    MaskMng.ValueWasChanged:= TRUE;
                12:(*Analog inputs*)
                    IF (Display.En_RealValue[1]) THEN
                        Display.value_REAL[1]:= Display.value_REAL[1] - TO_REAL(__SYSVA_KEY_COUNTER)/10.0;
                        IF (Display.value_REAL[1] < Display.value_MinREAL[1]) THEN
                            Display.value_REAL[1]:= Display.value_MaxREAL[1];
                            __SYSVA_KEY_COUNTER:= 0;
                            Beep();
                        END_IF;
                    ELSIF (Display.En_IntValue[1]) THEN
                        Display.value_INT[1]:= Display.value_INT[1] - TO_INT(__SYSVA_KEY_COUNTER)/10 - 1;
                        IF (Display.value_INT[1] < Display.value_MinINT[1]) THEN
                            Display.value_INT[1]:= Display.value_MaxINT[1];
                            __SYSVA_KEY_COUNTER:= 0;
                            Beep();
                        END_IF;
                    END_IF;
                    //MaskMng.ValueWasChanged:= TRUE;

                14:
                    Display.value_REAL[1]:= Display.value_REAL[1] - TO_REAL(__SYSVA_KEY_COUNTER)/10.0;
                    IF (Display.value_REAL[1] < 0.0) THEN
                        Display.value_REAL[1]:= 0.0;
                        Beep();
                    END_IF;
            END_CASE;
        ELSIF (CurRow_modePRG = 5) THEN // Изменение инверсии
            IF (Display.value_BOOL[3] = 0) THEN
                Display.value_BOOL[3]:= 1;
            ELSE
                Display.value_BOOL[3]:= 0;
            END_IF;
        END_IF;
    ELSE
        mask_List_pos:=  mask_List_pos + TO_DINT(__SYSVA_KEY_COUNTER)/20 + 1;
        IF (mask_List_pos > cnt_Items) THEN
            __SYSVA_KEY_COUNTER:= 0;
            mask_List_pos:= 1;
            Beep();
        END_IF;
        Display.Descr[1]:= TO_UINT(cfgIO.Link_toCodes[TO_DINT(mask_List[mask_List_pos])]) - TO_UINT(MaskMng.sig_start) + 1;
        Display.Descr[2]:= mask_List[mask_List_pos];
    END_IF;
END_FUNCTION

FUNCTION IO_UP
    IF (StatePRG = STATE_PRG_ON) THEN
        IF (CurRow = 3) THEN // Надпись Режим
            IF (Display.value_BOOL[1] = 1) THEN //руч.
                CurRow:= 4;
            ELSE
                IF  (Display.MaskID = 11) OR // Дискретные входы
                    (Display.MaskID = 14)    // Аналоговые выходы
                THEN
                    CurRow:= 5;
                ELSE
                    Beep();
                END_IF;
            END_IF;
        ELSIF (CurRow = 4) THEN // Надпись Статус
            CurRow:= 3;
        ELSIF (CurRow = 5) THEN // Надпись инверсия
            CurRow:= 3;
        ELSIF (CurRow_modePRG = 3) THEN // Изменение режима
            IF (Display.value_BOOL[1] = 0) THEN
                 Display.value_BOOL[1]:= 1;
            ELSIF( Display.value_BOOL[1] = 1) THEN
                Display.value_BOOL[1]:= 0;
            END_IF;
            //MaskMng.ValueWasChanged:= TRUE;
        ELSIF (CurRow_modePRG = 4) THEN // Изменение значения
            CASE Display.MaskID OF
                11, 13:(*Digital*)
                    Display.value_BOOL[2]:= 1; //ON
                    MaskMng.ValueWasChanged:= TRUE;
                12:(*Analog inputs*)
                    IF (Display.En_RealValue[1]) THEN
                        Display.value_REAL[1]:= Display.value_REAL[1] + TO_REAL(__SYSVA_KEY_COUNTER)/10.0;
                        IF (Display.value_REAL[1] > Display.value_MaxREAL[1]) THEN
                            Display.value_REAL[1]:= Display.value_MinREAL[1];
                            __SYSVA_KEY_COUNTER:= 0;
                            Beep();
                        END_IF;
                    ELSIF (Display.En_IntValue[1]) THEN
                        Display.value_INT[1]:= Display.value_INT[1] + TO_INT(__SYSVA_KEY_COUNTER)/10 + 1;
                        IF (Display.value_INT[1] > Display.value_MaxINT[1]) THEN
                            Display.value_INT[1]:= Display.value_MinINT[1];
                            __SYSVA_KEY_COUNTER:= 0;
                            Beep();
                        END_IF;
                    END_IF;

                14: (*Analog outputs*)
                    Display.value_REAL[1]:= Display.value_REAL[1] + TO_REAL(__SYSVA_KEY_COUNTER)/10.0;
                    IF (Display.value_REAL[1] > 10.0) THEN
                        Display.value_REAL[1]:= 10.0;
                        Beep();
                    END_IF;
            END_CASE;
        ELSIF (CurRow_modePRG = 5) THEN // Изменение инверсии
            IF (Display.value_BOOL[3] = 1) THEN
                Display.value_BOOL[3]:= 0;
            ELSE
                Display.value_BOOL[3]:= 1;
            END_IF;
        END_IF;
    ELSE
        mask_List_pos:=  mask_List_pos - TO_DINT(__SYSVA_KEY_COUNTER)/20 - 1;
        IF (mask_List_pos < 1) THEN
            __SYSVA_KEY_COUNTER:= 0;
            mask_List_pos:= cnt_Items;
            Beep();
        END_IF;
        Display.Descr[1]:= TO_UINT(cfgIO.Link_toCodes[TO_DINT(mask_List[mask_List_pos])]) - TO_UINT(MaskMng.sig_start) + 1;
        Display.Descr[2]:= mask_List[mask_List_pos];
    END_IF;
END_FUNCTION

FUNCTION IO_PRG
    IF (StatePRG = STATE_PRG_READY) THEN        // вход в режим редактирования
        StatePRG:=  STATE_PRG_ON;
        CurRow:= 3;
        CurRow_modePRG:= 0;
    ELSIF (StatePRG = STATE_PRG_ON) THEN        // выход из режима редактирования
        StatePRG:=  STATE_PRG_READY;
        CurRow:= 0;
        CurRow_modePRG:= 0;
        MaskMng.ValueWasChanged:= TRUE;
    ELSIF (StatePRG = STATE_PRG_OFF) THEN        //ручной режим недоступен
        ShowPopUpMessage(17, SHORT_POPUP_TIME);
    END_IF;
END_FUNCTION

FUNCTION IO_ENTER
     IF (StatePRG = STATE_PRG_ON) THEN  // ручное управление
        IF (CurRow <> 0) THEN           // Пункты
           // IF (mask_List[mask_List_pos] >= 64) AND (mask_List[mask_List_pos] <= 83) THEN
            //    Beep();
            //ELSE          // НЕ DP-TOP
                CurRow_modePRG:= CurRow;
                CurRow:= 0;
           // END_IF;
        ELSIF (CurRow_modePRG = 3) THEN // Режим
            CurRow:= CurRow_modePRG;
            CurRow_modePRG:= 0;
            MaskMng.ValueWasChanged:= TRUE;
        ELSIF (CurRow_modePRG = 4) THEN // Статус
            CurRow:= CurRow_modePRG;
            CurRow_modePRG:= 0;
            MaskMng.ValueWasChanged:= TRUE;
        ELSIF (CurRow_modePRG = 5) THEN // Инверсия
            CurRow:= CurRow_modePRG;
            CurRow_modePRG:= 0;
            MaskMng.ValueWasChanged:= TRUE;
        END_IF;
    END_IF;
END_FUNCTION
//---------------------------------------------------------------

// Управление маской коррекции -------------------------------------
FUNCTION CORR_DOWN

    IF (StatePRG = STATE_PRG_ON) THEN
        (*Analog inputs correction*)
        IF (Display.En_RealValue[1]) THEN
            //Display.value_REAL[1]:= Display.value_REAL[1] - TO_REAL(__SYSVA_KEY_COUNTER)/10.0;
            Display.value_REAL[1]:= Display.value_REAL[1] - Display.value_REAL[8];
            IF (Display.value_REAL[1] < Display.value_MinREAL[1]) THEN
                Display.value_REAL[1]:= Display.value_MaxREAL[1];
                __SYSVA_KEY_COUNTER:= 0;
                Beep();
            END_IF;
        ELSIF (Display.En_IntValue[1]) THEN
            //Display.value_INT[1]:= Display.value_INT[1] - TO_INT(__SYSVA_KEY_COUNTER)/10 - 1;
            Display.value_INT[1]:= Display.value_INT[1] - Display.value_INT[8];
            IF (Display.value_INT[1] < Display.value_MinINT[1]) THEN
                Display.value_INT[1]:= Display.value_MaxINT[1];
                __SYSVA_KEY_COUNTER:= 0;
                Beep();
            END_IF;
        END_IF;
    ELSE
        mask_List_pos:=  mask_List_pos + TO_DINT(__SYSVA_KEY_COUNTER)/20 + 1;
        IF (mask_List_pos > cnt_Items) THEN
            __SYSVA_KEY_COUNTER:= 0;
            mask_List_pos:= 1;
            Beep();
        END_IF;
        Display.Descr[1]:= TO_UINT(cfgIO.Link_toCodes[TO_DINT(mask_List[mask_List_pos])]) - TO_UINT(MaskMng.sig_start) + 1;
        Display.Descr[2]:= mask_List[mask_List_pos];
    END_IF;

END_FUNCTION

FUNCTION CORR_UP

    IF (StatePRG = STATE_PRG_ON) THEN
        (*Analog inputs correction*)
        IF (Display.En_RealValue[1]) THEN
            //Display.value_REAL[1]:= Display.value_REAL[1] + TO_REAL(__SYSVA_KEY_COUNTER)/10.0;
            Display.value_REAL[1]:= Display.value_REAL[1] + Display.value_REAL[8];
            IF (Display.value_REAL[1] > Display.value_MaxREAL[1]) THEN
                Display.value_REAL[1]:= Display.value_MinREAL[1];
                __SYSVA_KEY_COUNTER:= 0;
                Beep();
            END_IF;
        ELSIF (Display.En_IntValue[1]) THEN
            //Display.value_INT[1]:= Display.value_INT[1] + TO_INT(__SYSVA_KEY_COUNTER)/10 + 1;
            Display.value_INT[1]:= Display.value_INT[1] + Display.value_INT[8];
            IF (Display.value_INT[1] > Display.value_MaxINT[1]) THEN
                Display.value_INT[1]:= Display.value_MinINT[1];
                __SYSVA_KEY_COUNTER:= 0;
                Beep();
            END_IF;
        END_IF;
    ELSE
        mask_List_pos:=  mask_List_pos - TO_DINT(__SYSVA_KEY_COUNTER)/20 - 1;
        IF (mask_List_pos < 1) THEN
            __SYSVA_KEY_COUNTER:= 0;
            mask_List_pos:= cnt_Items;
            Beep();
        END_IF;
        Display.Descr[1]:= TO_UINT(cfgIO.Link_toCodes[TO_DINT(mask_List[mask_List_pos])]) - TO_UINT(MaskMng.sig_start) + 1;
        Display.Descr[2]:= mask_List[mask_List_pos];
    END_IF;

END_FUNCTION

FUNCTION CORR_PRG
    IF (StatePRG = STATE_PRG_READY) THEN        // вход в режим редактирования
        StatePRG:=  STATE_PRG_ON;
        CurRow:= 0;
        CurRow_modePRG:= 3;
    ELSIF (StatePRG = STATE_PRG_ON) THEN        // выход из режима редактирования
        StatePRG:=  STATE_PRG_READY;
        CurRow:= 0;
        CurRow_modePRG:= 0;
        MaskMng.ValueWasChanged:= TRUE;
    ELSIF (StatePRG = STATE_PRG_OFF) THEN        //ручной режим недоступен
        ShowPopUpMessage(17, SHORT_POPUP_TIME);
    END_IF;
END_FUNCTION

FUNCTION CORR_ENTER
    IF (StatePRG = STATE_PRG_ON) THEN  // ручное управление
        MaskMng.ValueWasChanged:= TRUE;
    END_IF;
END_FUNCTION
//---------------------------------------------------------------
//----------------------- Main Menu -----------------------------
FUNCTION MainMenu_DOWN   // Переход вниз

    IF (CurRow < num_Rows) THEN
        Display.UoM[CurRow]:= Display.UoM[CurRow] - 1;
        CurRow:= CurRow + 1;
        Display.UoM[CurRow]:= Display.UoM[CurRow] + 1;
    ELSE
        Position:= Position + TO_DINT(__SYSVA_KEY_COUNTER)/20 + 1;

        IF (Position > cnt_Items - num_Rows + 1) THEN
            __SYSVA_KEY_COUNTER:= 0;
            Position:= 1;
            CurRow:= 1;
            //Beep();
        END_IF;
        update_MainMenu_List:= TRUE;
    END_IF;

    CurList_Position:= Position + CurRow - 1;
END_FUNCTION

FUNCTION MainMenu_UP   // Переход вверх

    IF (CurRow > 1) THEN
        Display.UoM[CurRow]:= Display.UoM[CurRow] - 1;
        CurRow:= CurRow - 1;
        Display.UoM[CurRow]:= Display.UoM[CurRow] + 1;
    ELSE
        Position:= Position - TO_DINT(__SYSVA_KEY_COUNTER)/20 - 1;

        IF (Position < 1) THEN
            __SYSVA_KEY_COUNTER:= 0;
            Position:= cnt_Items - num_Rows + 1;
            CurRow:= num_Rows;
            //Beep();
        END_IF;
        update_MainMenu_List:= TRUE;
    END_IF;

    CurList_Position:= Position + CurRow - 1;
END_FUNCTION

FUNCTION MainMenu_ENTER   //

    IF (Display.value_Type[CurRow] = 0) // каталог
    THEN
        IF (CurLevel < 10) THEN
            SaveMenuPos();
            //CurLevel:= CurLevel + 1;
            CurMenuPoint:= TO_DINT(Display.Descr[CurRow]);
            getMainMenu:= TRUE;
        END_IF;
        CurRow:= 1;
        Position:= 1;
    ELSIF (Display.value_Type[CurRow] = 1) // переход на  другую маску
    THEN
        //CurMenuPoint:= Display.Descr[CurRow];
        //getMainMenu:= TRUE;
        SaveMenuPos();
        //CurLevel:= CurLevel + 1;
        GotoMaskID(TO_USINT(Display.value_MinINT[CurRow]), TO_USINT(Display.value_MaxINT[CurRow]));
        Display.UoM[1]:= 0;
        Display.UoM[2]:= 0;
        Display.UoM[3]:= 0;
        Display.Descr[1]:= 0;
        Display.Descr[2]:= 0;
        Display.Descr[3]:= 0;
        CurRow:= 0;
    ELSIF (Display.value_Type[CurRow] = 2) // всплывающие окна
    THEN
        SaveMenuPos();
        GotoMaskID(TO_USINT(Display.value_MinINT[CurRow]), TO_USINT(Display.value_MaxINT[CurRow]));
    END_IF;
    CurList_Position:= 1;
END_FUNCTION

FUNCTION MainMenu_ESC   //
    IF (CurLevel > 1) THEN
        LoadMenuPos();
        getMainMenu:= TRUE;
    ELSE
        GlobalEsc();
    END_IF;
END_FUNCTION

//---------------------------------------------------------------
FUNCTION GotoMaskID
//Загрузка маски или петли по MaskID с сохранением пути
    VAR_INPUT
        iMaskID : USINT;
    END_VAR

    StoreMaskID();
    LoadMaskID(iMaskID, 0);
END_FUNCTION

FUNCTION GotoMaskID
//Загрузка маски или петли по MaskID с сохранением пути
    VAR_INPUT
        iMaskID : USINT;
        iParam : USINT; // передаваемый параметр
    END_VAR

    StoreMaskID();
    LoadMaskID(iMaskID, iParam);
END_FUNCTION

FUNCTION LoadMaskID
//Загрузка маски или петли по MaskID
    VAR_INPUT
        iMaskID : USINT;
        iParam : USINT; // передаваемый параметр
    END_VAR

    Display.MaskID:= TO_UINT(iMaskID);

    CASE iMaskID OF
        1: // Гл.экран	DF_MID_MAIN
            //GotoLoop(MAIN);
            GotoMask(Main_Mask);
            //При выходе в гл.меню или на гл.экран система возвращается в работу
            SystemPause:= FALSE;

        2: // Логин	DF_MID_LOGIN
            PwdIn := 0;                 // Reset password
            IncrTmp := 0;
            PwdRes := 0;
            CleanPwd();
            GotoMask(Pwd_LogIn);

        3: // Осн.меню	DF_MID_MMENU
            MainMenuVisibility_Is_Set:= FALSE;
	        ParamVisibility_Is_Set:= 	FALSE;

            getMainMenu:= TRUE;
            StatePRG:= STATE_PRG_OFF;
            GotoMask(Menu_Main);
            //При выходе в гл.меню или на гл.экран система вовзвращается в работу
            SystemPause:= FALSE;

        4: // Управление	DF_MID_ONOFF
            IF (LocalMode = 0)AND(Role_Slave) THEN
                StatePRG:= STATE_PRG_READY;// режим до редактирования
            ELSE
                StatePRG:= STATE_PRG_ALWAYS_ON;// режим редактирования
            END_IF;
            GotoLoop(ONOFF);

        5: // Маска загрузки	DF_MID_LOAD
            IF (UnitOff) THEN
                MaskMng.LoadMaskMode:= iParam;

                IF (iParam = 0) THEN //Загрузка при выходе из конфигуратора
                    ConfigMng.checkConfigFile:= TRUE;
                ELSIF (iParam = 1) THEN //Загрузка при входе в конфигуратор
                    ConfigMng.checkConfigFile:= TRUE;
                ELSIF (iParam = 2) THEN   //Загрузка конфигуратора из конфигуратора
                    //CurLevel:= ConfigStartLevel; возвращаемся к началу конфигуратора
                    //CurList_Position:= 1;
                   IsConfigChanged:= TRUE;
                    load_Config:= TRUE;
                ELSIF (iParam = 3) THEN   //Сохранение конфигуратора без выхода
                    save_Config:= TRUE;
                ELSIF (iParam = 4) THEN   //Сохранение конфигуратора с выходом
                    save_Config:= TRUE;
                END_IF;

                GotoMask(LoadConfig_Mask);
            ELSE
                ShowPopUpMessage(1, POPUP_TIME, TRUE);//  Выключите установку для изменения настроек!
            END_IF;
        6: //Настройки Ethernet DF_MID_ETH
            read_EthernetSettings:= TRUE;
            StatePRG:= STATE_PRG_READY;
            GotoMask(EthernetConfig_Mask);

        7: // Управление расписанием	DF_MID_SCH_MG
            temp_En_Schedule:= En_Schedule;
            StatePRG:= STATE_PRG_ON;
            GotoMask (Schedule_Manage);

        8: // Журнал аварий	DF_MID_ALOG
            gotoAlarmLog();

        9: // Последовательности	DF_MID_SEQ
            GotoLoop(SEQUENCES);

        10: // Мастер конфигурации	DF_MID_CFG_M
            IF (iParam = 1) THEN
                CurMenuPoint:=  0;
                Position:= 1;
                CurList_Position:= 1;
                CurRow:= 1;
                CurRow_modePRG:=    0;
                ConfigStartLevel:= CurLevel;
            END_IF;

            getConfigMenu:= TRUE;
            GotoMask(REF_CONFIGURATOR);

        11: //Дискретные входы	DF_MID_IO_DI
            CurRow:=            1;
            CurRow_modePRG:=    0;
            getIOList:=         TRUE;
            IF (UnitOn) THEN
                StatePRG:= STATE_PRG_OFF;
            ELSE
                StatePRG:= STATE_PRG_READY;
            END_IF;
            GotoMask(IO_DI);

        12: //Аналоговые входы	DF_MID_IO_AI
            CurRow:=            1;
            CurRow_modePRG:=    0;
            getIOList:=         TRUE;
            IF (UnitOn) THEN
                StatePRG:= STATE_PRG_OFF;
            ELSE
                StatePRG:= STATE_PRG_READY;
            END_IF;
            GotoMask(IO_AI);

        13: //Дискретные выходы	DF_MID_IO_DO
            CurRow:=            1;
            CurRow_modePRG:=    0;
            getIOList:=         TRUE;
            IF (UnitOn) THEN
                StatePRG:= STATE_PRG_OFF;
            ELSE
                StatePRG:= STATE_PRG_READY;
            END_IF;
            GotoMask(IO_DO);

        14: //Аналоговые выходы	DF_MID_IO_AO
            CurRow:=            1;
            CurRow_modePRG:=    0;
            getIOList:=         TRUE;
            IF (UnitOn) THEN
                StatePRG:= STATE_PRG_OFF;
            ELSE
                StatePRG:= STATE_PRG_READY;
            END_IF;
            GotoMask(IO_AO);

        15: //Уставка	DF_MID_SET
            getParam:= TRUE;
            IF (LocalMode = 0)AND(Role_Slave) THEN
                StatePRG:= STATE_PRG_READY;// режим до редактирования
            ELSE
                StatePRG:= STATE_PRG_ALWAYS_ON;// режим редактирования
            END_IF;
            GotoLoop(SET);

        16: //Выход	DF_MID_OUT
            GotoMask(Pwd_LogOut);

        17: //Роль устройства	DF_MID_GROLE
            temp_Role:= Role;
            StatePRG:= STATE_PRG_ALWAYS_ON;
            Gotomask(DeviceRole);
            GotoCursor (0,10);// кидаем за пределы экрана. ТОЛЬКО ДЛЯ 1 IO переменной на экране! Использовать Compare() без NextField!

        18: //Настройки группы	DF_MID_GSET
            IF (Role_Master) THEN
                IF (Num_Slaves > 0) THEN
                    CurSlave:=  1;
                    CurSlaveShow:=  TRUE;
                    StatePRG:= STATE_PRG_READY;// режим готовности к редактированию
                    GotoMask (SlaveSet);
                ELSE
                    ShowPopUpMessage(6, POPUP_TIME, TRUE);//  Состав группы не объявлен!
                END_IF;
            ELSE
                StatePRG:= STATE_PRG_ON;// режим готовности к редактированию
                Gotomask(LocalSet);// если ведомый - местные настройки (выбор режима)
                GotoCursor(0,10);
            END_IF;

        19: //Состав группы	DF_MID_GSTCT
            IF (Role_Master) THEN
                StatePRG:= STATE_PRG_ALWAYS_ON;// режим редактирования сразу
                Gotomask(GroupStructure);// если мастер-переходим к выбору состава группы
                GotoCursor (0,10);// кидаем за пределы экрана. ТОЛЬКО ДЛЯ 1 IO переменной на экране! Использовать Compare() без NextField!
           ELSE
                ShowPopUpMessage(2, POPUP_TIME, TRUE);//  Для доступа, выберите роль устройства: ВЕДУЩИЙ // если ведомый - заглушка
           END_IF;

        20: // Маска параметров	DF_MID_PAR
            //setParamMask(TO_USINT(Display.value_MaxINT[CurRow]));
            CurParam:=          iParam;
            getParamMenu:=      TRUE;
            cnt_Items:=         0;
            StatePRG:=          STATE_PRG_READY;
            GotoMask(REF_Parameters);

        21: //ХМ: Статистика	DF_MID_CM_STA
            //Show_CompStats:= TRUE;
            Display.Index:=     -1;
            StatePRG:=          STATE_PRG_READY;
            GotoLoop(FRIDGE_STATS);

        22: // Дата и время	DF_MID_DTIME
            StatePRG:=          STATE_PRG_READY;
            GotoLoop(DATETIME);

        23: //Язык	DF_MID_LANG
            StatePRG:=          STATE_PRG_ALWAYS_ON;
            Gotomask(Language);

        24: //Управление доступом	DF_MID_PASS
            IncrTmp :=          0;
            StatePRG:=          STATE_PRG_READY;
            GotoMask(PWDCHG);

        25: //Коррекция датчиков	DF_MID_SCORR
            MaskMng.getCorrList:= TRUE;
            StatePRG:= STATE_PRG_READY;
            GotoMask(CORR_AI);

        26: //Настройки ModBus	DF_MID_MODBUS
            IF (is_TOP) THEN
                ShowPopUpMessage(9, POPUP_TIME, TRUE);//  Доступно только со шкафа управления!
            // 20.07.20 v.2.6.0.0
            //ELSIF (IsDLE)AND(Role_Slave) THEN
            //    ShowPopUpMessage(10, POPUP_TIME, TRUE);//  Доступно только с ВЕДУЩЕГО!
            ELSE
                IF (Ethernet.Protocol[1] = 4) OR (Ethernet.Protocol[1] = 5) THEN
                    MB_port:= 1;
                ELSIF (BMS_card.Protocol = 4) OR (BMS_card.Protocol = 5) THEN
                    MB_port:= 2;
                ELSIF (BMS2.Protocol = 4) OR (BMS2.Protocol = 5) THEN
                    MB_port:= 3;
                ELSE
                    MB_port:= 0;
                END_IF;
                Temp_MB_port:= MB_port;
                Temp_MB_Address:= MB_Address;
                Show_ports();
                StatePRG:= STATE_PRG_READY;
                GotoLoop(MODBUS);
            END_IF;

        27: //Обновление	DF_MID_UPGR
            IF (UnitOff) THEN
                IF (iParam = 1) THEN //USB
                    IF (isUSB) THEN
                        Upgrade.UpgradeDrive:= 1; //SYS_DISK_USB
                        Upgrade.Check_Upgrade:= TRUE;
                        StatePRG:= STATE_PRG_ALWAYS_ON;
                        NextCycleAction:= 4; // GotoLoop (UPGRADE);
                    ELSE
                        //Вставьте USB-накопитель
                        ShowPopUpMessage(24, SHORT_POPUP_TIME, TRUE);
                    END_IF;
                ELSE
                    Upgrade.UpgradeDrive:= 0; //SYS_DISK_INTERNAL
                    Upgrade.Check_Upgrade:= TRUE;
                    StatePRG:= STATE_PRG_ALWAYS_ON;
                    NextCycleAction:= 4; // GotoLoop (UPGRADE);
                END_IF;
            ELSE
                ShowPopUpMessage(1, POPUP_TIME, TRUE);//  Выключите установку для изменения настроек!
            END_IF;

        28: //Расписание	DF_MID_SCH
            IF (is_TOP) THEN
                ShowPopUpMessage(9, POPUP_TIME, TRUE);//  Доступно только со шкафа управления!
            ELSIF (IsDLE)AND(Role_Slave) THEN
                ShowPopUpMessage(10, POPUP_TIME, TRUE);//  Доступно только с ВЕДУЩЕГО!
            ELSE
                StatePRG:= STATE_PRG_READY;
                GotoLoop (SCHEDULE);
            END_IF;

        29: //Режим управления	DF_MID_CMOD
            IF (is_TOP) THEN
                ShowPopUpMessage(9, POPUP_TIME, TRUE);//  Доступно только со шкафа управления!
            ELSIF (IsDLE)AND(Role_Slave)AND NOT(LocalMode) THEN
                ShowPopUpMessage(10, POPUP_TIME, TRUE);//  Доступно только с ВЕДУЩЕГО!
            ELSE
                temp_Mode_Control:= Mode_Control;
                StatePRG:= STATE_PRG_ON;
                GotoLoop (CONTROL_MODE);
            END_IF;

        30: //Маска сообщения	DF_MID_MSG
            ;

        31: //Маска вопроса	DF_MID_QSTN
            ReturnToPrevMask:= TRUE;
            StatePRG:= STATE_PRG_OFF;
            DTPopUp:= 0; //без таймера всплывающего окна
            PopUp_Question:= iParam;
            Gotomask(PopUp_Question_Mask);

        32: //Маска ведомых   DF_MID_SLST
            MaskMng.setStatePRG:= TRUE;
            GotoLoop(SLAVESTATES);

        33: //Роль устройства	DF_MID_ROLE
            temp_Role:= Role;
            StatePRG:= STATE_PRG_ALWAYS_ON;// режим редактирования сразу
            GotoLoop(UNITCONFIG);
            GotoCursor (0,10);// кидаем за пределы экрана. ТОЛЬКО ДЛЯ 1 IO переменной на экране! Использовать Compare() без NextField!

        34: //Настройки BMS   DF_MID_BMS
            IF (Role_Slave)OR(is_TOP) THEN
                Temp_MB_Baudrate:= BMS2.Baudrate;
                Temp_MB_Parity:= BMS2.Parity;
                Temp_MB_StopBits:= BMS2.StopBits;
            ELSE
                Temp_MB_Baudrate:= FBus2.Baudrate;
                Temp_MB_Parity:= FBus2.Parity;
                Temp_MB_StopBits:= FBus2.StopBits;
            END_IF;
            En_MB_BMS:= TRUE;
            StatePRG:= STATE_PRG_READY;//
            GotoLoop(BMS_SETTINGS);

         35: //Загрузка/Сохранение на USB DF_MID_PARMNG
            IF (isUSB) THEN
                Display.Hint:= TO_UINT(iParam);
                IF (iParam = 1) THEN
                    ShowPopUpQuestion(23, TRUE); //Сохранить параметры на USB?
                ELSE
                    ShowPopUpQuestion(22, TRUE); //Загрузить параметры с USB?
                END_IF;
            ELSE
                ShowPopUpMessage(24, SHORT_POPUP_TIME, TRUE); //Вставьте USB-накопитель
            END_IF;

         36: //Дискретные входы (конфиг) DF_MID_CFG_DI
            Position:= 1;
            CurRow:= 1;
            cnt_Items:= 0;
            getIOConfig:= TRUE;

            GotoMask(CFG_DI);

         37: //Аналоговые входы (конфиг) DF_MID_CFG_AI
            Position:= 1;
            CurRow:= 1;
            cnt_Items:= 0;
            getIOConfig:= TRUE;

            GotoMask(CFG_AI);

         38: //Дискретные выходы (конфиг) DF_MID_CFG_DO
            Position:= 1;
            CurRow:= 1;
            cnt_Items:= 0;
            getIOConfig:= TRUE;

            GotoMask(CFG_DO);

         39: //Аналоговые выходы (конфиг) DF_MID_CFG_AO
            Position:= 1;
            CurRow:= 1;
            cnt_Items:= 0;
            getIOConfig:= TRUE;

            GotoMask(CFG_AO);

         40: //Холодильная машина DF_MID_COLM
            StatePRG:= STATE_PRG_OFF;
            GotoLoop(FRIDGE);

         41: //Карта сети DF_MID_NETM
            StatePRG:= STATE_PRG_OFF;
            IF (Role_Master) THEN // для мастера
                IF (Num_Slaves > 0) THEN
                    Gotomask(NetMap);
                    IF (CurPosition = 0)OR(CurPosition > Num_Slaves) THEN
                        CurPosition:=   1;// в первую позицию, если впервые. Остальные запоминаем
                    END_IF;
                    CurShow[CurPosition]:=  TRUE;
                ELSE
                    ShowPopUpMessage(6, POPUP_TIME); //Состав группы не объявлен!
                END_IF;
            ELSE // для ведомых
                Gotomask(MasterState);
            END_IF;

        42: //Информация DF_MID_INFO
            GotoLoop(INFO);

        43: //Набор уставок	DF_MID_PSET
            getParam:= TRUE;
            StatePRG:= STATE_PRG_ALWAYS_ON;// режим редактирования
            GotoLoop(PRESETS);
            GotoCursor(0, 10);

        44: //Пароувлажнитель DF_MID_HUMID
            GotoLoop(HUMID);

        45: //Настройки соединения DF_MID_RESSET
            StatePRG:=              STATE_PRG_READY;
            MaskMng.get_Slave_IP:=  TRUE;
            GotoLoop(RES_SLAVE_SETTINGS);

    END_CASE;
END_FUNCTION

FUNCTION StoreMaskID
//Сохраняем позицию маски
    MaskIDStore[MaskIDLevel]:= TO_USINT(Display.MaskID);
    IF (MaskIDLevel < 9) THEN
        MaskIDLevel:= MaskIDLevel + 1;
    END_IF;
END_FUNCTION

FUNCTION ReStoreMaskID
//Загружаем позицию маски
    IF (MaskIDLevel > 0) THEN
        MaskIDLevel:= MaskIDLevel - 1;
    END_IF;
    Display.MaskID:= TO_UINT(MaskIDStore[MaskIDLevel]);
    MaskIDStore[MaskIDLevel]:= 0;
    LoadMaskID(TO_USINT(Display.MaskID), 0);
END_FUNCTION

FUNCTION SaveMenuPos
//Сохраняем состояние меню
    Display.Path.MenuPoint[CurLevel]:=  CurMenuPoint;
    Display.Path.Position[CurLevel]:=   Position;
    Display.Path.Row[CurLevel]:=        CurRow;
    Display.Path.Row_PRG[CurLevel]:=    CurRow_modePRG;

    IF (CurRow = 0) AND (CurRow_modePRG <> 0) THEN
        CurMenuPoint:= TO_DINT(Display.Descr[CurRow_modePRG]);
    ELSIF (CurRow <> 0) THEN
        CurMenuPoint:= TO_DINT(Display.Descr[CurRow]);
    END_IF;

    IF (CurLevel < 10) THEN
        CurLevel:= CurLevel + 1;
    ELSE
         CurLevel:= 10;
    END_IF;
END_FUNCTION

FUNCTION LoadMenuPos
//Загружаем состояние меню
    IF (CurLevel > 0) THEN
        CurLevel:= CurLevel - 1;
    ELSE
         CurLevel:= 0;
    END_IF;

    CurMenuPoint:=      Display.Path.MenuPoint[CurLevel];
    Position:=          Display.Path.Position[CurLevel];
    CurRow:=            Display.Path.Row[CurLevel];
    CurRow_modePRG:=    Display.Path.Row_PRG[CurLevel];
    CurList_Position:=  Position + CurRow - 1;

    Display.Path.MenuPoint[CurLevel]:=      0;
    Display.Path.Position[CurLevel]:=       0;
    Display.Path.Row[CurLevel]:=         0;
    Display.Path.Row_PRG[CurLevel]:= 0;
END_FUNCTION

FUNCTION ClearHistory
//Очистка истории
    MaskIDLevel:= 0;
    MaskIDStore[0]:= 0;
    MaskIDStore[1]:= 0;
    MaskIDStore[2]:= 0;
    MaskIDStore[3]:= 0;
    MaskIDStore[4]:= 0;
    MaskIDStore[5]:= 0;
    MaskIDStore[6]:= 0;
    MaskIDStore[7]:= 0;
    MaskIDStore[8]:= 0;
    MaskIDStore[9]:= 0;
    Position:= 0;
    CurRow:= 0;
    CurList_Position:= 0;

    CurLevel:= 0;
    Display.Path.MenuPoint[0]:= 0;
    Display.Path.Position[0]:= 0;
    Display.Path.Row[0]:= 0;
    Display.Path.MenuPoint[1]:= 0;
    Display.Path.Position[1]:= 0;
    Display.Path.Row[1]:= 0;
    Display.Path.MenuPoint[2]:= 0;
    Display.Path.Position[2]:= 0;
    Display.Path.Row[2]:= 0;
    Display.Path.MenuPoint[3]:= 0;
    Display.Path.Position[3]:= 0;
    Display.Path.Row[3]:= 0;
    Display.Path.MenuPoint[4]:= 0;
    Display.Path.Position[4]:= 0;
    Display.Path.Row[4]:= 0;
    Display.Path.MenuPoint[5]:= 0;
    Display.Path.Position[5]:= 0;
    Display.Path.Row[5]:= 0;
    Display.Path.MenuPoint[6]:= 0;
    Display.Path.Position[6]:= 0;
    Display.Path.Row[6]:= 0;
    Display.Path.MenuPoint[7]:= 0;
    Display.Path.Position[7]:= 0;
    Display.Path.Row[7]:= 0;
    Display.Path.MenuPoint[8]:= 0;
    Display.Path.Position[8]:= 0;
    Display.Path.Row[8]:= 0;
    Display.Path.MenuPoint[9]:= 0;
    Display.Path.Position[9]:= 0;
    Display.Path.Row[9]:= 0;
    Display.Path.MenuPoint[10]:= 0;
    Display.Path.Position[10]:= 0;
    Display.Path.Row[10]:= 0;

END_FUNCTION
FUNCTION Hide_Baudrate_Class_DOWN
    CASE __TMP_UDINT OF
        1200:
            Beep();
            __TMP_UDINT:= 375000;
        2400:
            __TMP_UDINT:= 1200;
        4800:
            __TMP_UDINT:= 2400;
        9600:
            __TMP_UDINT:= 4800;
        19200:
            __TMP_UDINT:= 9600;
        38400:
            __TMP_UDINT:= 19200;
        57600:
            __TMP_UDINT:= 38400;
        76800:
            __TMP_UDINT:= 57600;
        115200:
            __TMP_UDINT:= 76800;
        375000:
            __TMP_UDINT:= 115200;
    END_CASE;
END_FUNCTION

FUNCTION Hide_Baudrate_Class_UP
    CASE __TMP_UDINT OF
        1200:
            __TMP_UDINT:= 2400;
        2400:
            __TMP_UDINT:= 4800;
        4800:
            __TMP_UDINT:= 9600;
        9600:
            __TMP_UDINT:= 19200;
        19200:
            __TMP_UDINT:= 38400;
        38400:
            __TMP_UDINT:= 57600;
        57600:
            __TMP_UDINT:= 76800;
        76800:
            __TMP_UDINT:= 115200;
        115200:
            __TMP_UDINT:= 375000;
        375000:
            Beep();
            __TMP_UDINT:= 1200;
    END_CASE;
END_FUNCTION

FUNCTION Net_Settings_ESC
	IF (StatePRG = STATE_PRG_READY) THEN
        GlobalEsc();
    ELSIF (StatePRG = STATE_PRG_ON) THEN
        Compare();
        IF (Role_Slave) OR (is_TOP) THEN
            IF (Temp_MB_Baudrate <> BMS2.Baudrate) OR
                (Temp_MB_Parity <> BMS2.Parity) OR
                (Temp_MB_StopBits <> BMS2.StopBits)
                THEN
                ShowPopUpQuestion(20);// изменение настроек сети
            ELSE
                GlobalEsc();
            END_IF;
        ELSE
            IF (Temp_MB_Baudrate <> FBus2.Baudrate) OR
                (Temp_MB_Parity <> FBus2.Parity) OR
                (Temp_MB_StopBits <> FBus2.StopBits)
                THEN
                ShowPopUpQuestion(20);// изменение настроек сети
            ELSE
                GlobalEsc();
            END_IF;

        END_IF;
    END_IF;
END_FUNCTION

FUNCTION Net_Settings_PRG
	 IF (StatePRG = STATE_PRG_READY) THEN
        StoreMask();
        StatePRG:= STATE_PRG_ON;
        NextCycleAction:= 1;
    ELSIF (StatePRG = STATE_PRG_ON) THEN
        Compare();
        IF (Role_Slave) OR (is_TOP) THEN
            IF (Temp_MB_Baudrate <> BMS2.Baudrate) OR
                (Temp_MB_Parity <> BMS2.Parity) OR
                (Temp_MB_StopBits <> BMS2.StopBits)
                THEN
                ShowPopUpQuestion(20);// изменение настроек сети
            ELSE
                StatePRG:= STATE_PRG_READY;
                NextCycleAction:=   1;
            END_IF;

        ELSE
            IF (Temp_MB_Baudrate <> FBus2.Baudrate) OR
                (Temp_MB_Parity <> FBus2.Parity) OR
                (Temp_MB_StopBits <> FBus2.StopBits)
                THEN
                ShowPopUpQuestion(20);// изменение настроек сети
            ELSE
                StatePRG:= STATE_PRG_READY;
                NextCycleAction:=   1;
            END_IF;
        END_IF;
    END_IF;
END_FUNCTION

FUNCTION Stats_1_UP
    Display.Index:= Display.Index - 1;
    //IF (Display.Index > 1) THEN
        //Display.Index:= Display.Index - 1;
    //ELSE
        //Display.Index:= EQ_Cooler.CompNum;
    //END_IF;
END_FUNCTION

FUNCTION Stats_1_DOWN
    Display.Index:= Display.Index + 1;
    //IF (Display.Index < EQ_Cooler.CompNum) THEN
        //Display.Index:= Display.Index + 1;
    //ELSE
        //Display.Index:= 1;
    //END_IF;
END_FUNCTION

// сброс наработки компрессора
FUNCTION Stats_1_PRG
    IF (PwdTyp >= 2) THEN    // only if logged as service or manufacturer
        IF (Display.Index = 1) THEN
            ShowPopUpQuestion(8);// Сбросить статистику компрессора 1?
        ELSIF (Display.Index = 2) THEN
            ShowPopUpQuestion(9);// Сбросить статистику компрессора 2?
        ELSIF (Display.Index = 3) THEN
            ShowPopUpQuestion(10);// Сбросить статистику компрессора 3?
        END_IF;
    ELSE
        ShowPopUpMessage(4, POPUP_TIME);//  Введите Сервисный пароль для изменения Сервисных настроек
    END_IF;
END_FUNCTION

FUNCTION EthernetConfig_Mask_ESC
    IF (StatePRG = STATE_PRG_READY) THEN
        GlobalEsc();
    ELSIF (StatePRG = STATE_PRG_ON) THEN
        Compare();
	    ShowPopUpQuestion(6, TRUE); //Сохранить настройки Ethernet?
    END_IF;
END_FUNCTION

FUNCTION EthernetConfig_Mask_PRG

    IF (StatePRG = STATE_PRG_READY) THEN
        StoreMask();
        StatePRG:= STATE_PRG_ON;
    ELSIF (StatePRG = STATE_PRG_ON) THEN
        Compare();
	    write_EthernetSettings:= TRUE;
        StatePRG:= STATE_PRG_READY;
    END_IF;

    NextCycleAction:=   1;
END_FUNCTION

FUNCTION Res_Slave_Settings_Mask_ESC
    IF (StatePRG = STATE_PRG_READY) THEN
        GlobalEsc();
    ELSIF (StatePRG = STATE_PRG_ON) THEN
        Compare();
	    ShowPopUpQuestion(6, TRUE); //Сохранить настройки Ethernet?
    END_IF;
END_FUNCTION

FUNCTION Res_Slave_Settings_Mask_PRG

    IF (StatePRG = STATE_PRG_READY) THEN
        StoreMask();
        StatePRG:= STATE_PRG_ON;
    ELSIF (StatePRG = STATE_PRG_ON) THEN
        Compare();
	    MaskMng.setChanges:= TRUE;
        StatePRG:= STATE_PRG_READY;
    END_IF;

    NextCycleAction:=   1;
END_FUNCTION

FUNCTION Hide_DHCP_BOOL_SWAP_Class_ENTER
	IF NOT(Ethernet.DHCP) THEN
        GotoNextField();
    END_IF;
END_FUNCTION

FUNCTION Sequences_Mask_DOWN
    //Если есть куда двигаться и есть стрелка
    IF (Display.MaskHeader < 1) AND (Display.value_BOOL[7] <> 0) THEN
        Display.MaskHeader:= Display.MaskHeader + 1;
    END_IF;
END_FUNCTION

FUNCTION Sequences_Mask_UP
    //Если есть куда двигаться и есть стрелка
    IF (Display.MaskHeader > 0) AND (Display.value_BOOL[7] <> 0) THEN
        Display.MaskHeader:= Display.MaskHeader - 1;
    END_IF;
END_FUNCTION

FUNCTION Preset_PRG
    MaskMng.gotoParam:= TO_USINT(Display.value_INT[1]); //переходим в текущий набор
    CurList_Position:= 1;
END_FUNCTION

FUNCTION Preset_DOWN
    Display.value_INT[1]:= Display.value_INT[1] + TO_INT(__SYSVA_KEY_COUNTER)/20 + 1;;
	IF (Display.value_INT[1] > Display.value_MaxINT[1]) THEN
        Display.value_INT[1]:= Display.value_MinINT[1];
    END_IF;
    downArrow:= TRUE;
END_FUNCTION

FUNCTION Preset_UP
    Display.value_INT[1]:= Display.value_INT[1] - TO_INT(__SYSVA_KEY_COUNTER)/20 - 1;;
	IF (Display.value_INT[1] < Display.value_MinINT[1]) THEN
        Display.value_INT[1]:= Display.value_MaxINT[1];
    END_IF;
    upArrow:= TRUE;
END_FUNCTION

FUNCTION Preset_ENTER
	setParam:= TRUE;
END_FUNCTION

FUNCTION LoadMask // Функция для загрузки маски из стратегии
    IF (LoadMask.MaskID <> 0) THEN
        GotoMaskID(LoadMask.MaskID, LoadMask.Param);
        LoadMask.MaskID:=   0;
        LoadMask.Param:=    0;
    END_IF;
END_FUNCTION

FUNCTION Main_Mask_ESC //Функция перехода на следующий контроллер в pLAN сети
	IF(__SYSVA_KEY_COUNTER >= 2) THEN
        __SYSVA_KEY_COUNTER:= 0;
        ReleaseTerminal();
    END_IF;
END_FUNCTION

FUNCTION Main_Mask_ESC_DOWN //Функция перехода на следующий контроллер в pLAN сети
    ReleaseTerminal();
END_FUNCTION

FUNCTION Goto_FRIDGE_PARAMS //Переход к параметрах ХМ
    GotoMaskID(20, 10); //(DF_MID_PAR, DF_PRM_CM_PAR);
END_FUNCTION

FUNCTION Goto_FRIDGE_STATS //Переход к параметрах ХМ
    GotoMaskID(21,0); //DF_MID_CM_STA
END_FUNCTION

FUNCTION SwitchPGD
    SetKeySwitch(28);
END_FUNCTION
